SUBAPPLICATION Uebung_004a4 (* Toggle Flip-Flop mit IE mit BUTTON_SINGLE_CLICK mit E_SPLIT *)
  (* Standard: 61499-2; Description: Copyright (c) 2023 Meisterschulen am Ostbahnhof This program and the accompanying materials are made available under the terms of the Eclipse Public License 2.0 which is available at https://www.eclipse.org/legal/epl-2.0/ SPDX-License-Identifier: EPL-2.0 *)
  (* Version 1.0, 2023-10-23, Franz Höpfinger, Meisterschulen am Ostbahnhof *)
  PACKAGE Uebungen;
  IMPORT logiBUS::io::DI::logiBUS_DI::Input_I1;
  IMPORT logiBUS::io::DI::logiBUS_DI_Events::BUTTON_SINGLE_CLICK;
  IMPORT logiBUS::io::DQ::logiBUS_DO::Output_Q1;
  IMPORT logiBUS::io::DQ::logiBUS_DO::Output_Q2;
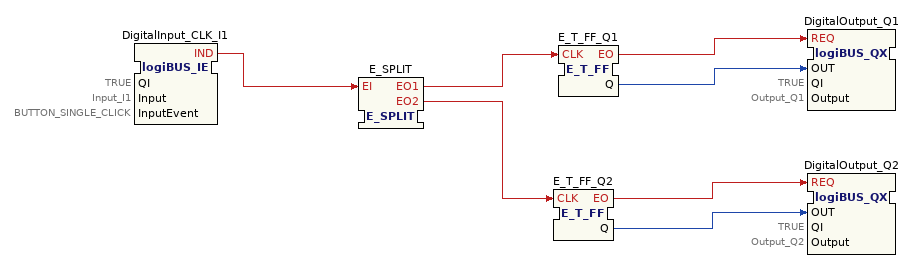
  (* hier 2x T_FF zu verwenden ist sinnlos, das soll nur zeigen wie man E_SPLIT verwenden kann. *)
  FBS
    DigitalOutput_Q1 : logiBUS::io::DQ::logiBUS_QX(QI := TRUE, Output := Output_Q1);
    DigitalInput_CLK_I1 : logiBUS::io::DI::logiBUS_IE(QI := TRUE, Input := Input_I1, InputEvent := BUTTON_SINGLE_CLICK);
    E_T_FF_Q1 : iec61499::events::E_T_FF;
    E_T_FF_Q2 : iec61499::events::E_T_FF;
    DigitalOutput_Q2 : logiBUS::io::DQ::logiBUS_QX(QI := TRUE, Output := Output_Q2);
    E_SPLIT : iec61499::events::E_SPLIT;
  END_FBS
  EVENT_CONNECTIONS
    E_T_FF_Q1.EO TO DigitalOutput_Q1.REQ;
    E_T_FF_Q2.EO TO DigitalOutput_Q2.REQ;
    E_SPLIT.EO1 TO E_T_FF_Q1.CLK;
    E_SPLIT.EO2 TO E_T_FF_Q2.CLK;
    DigitalInput_CLK_I1.IND TO E_SPLIT.EI;
  END_CONNECTIONS
  DATA_CONNECTIONS
    E_T_FF_Q1.Q TO DigitalOutput_Q1.OUT;
    E_T_FF_Q2.Q TO DigitalOutput_Q2.OUT;
  END_CONNECTIONS
END_SUBAPPLICATION
